// Interface handling generic data contained in a collection.
INTERFACE I_Generic_Collection EXTENDS I_Collection

END_INTERFACE

(* stored: Version 1.1.0.1, ProductVersion 3.1.4024.4
   Itf I_Generic_Collection: Id {882331ba-6be0-4573-976d-349fdb872347} *)
